PROGRAM MAIN
VAR
END_VAR

//Tc3_Motion.WareHousingExample_Tc3_DriveMotionControl();

WareHousingExample_Tc3_DriveMotionControl();

END_PROGRAM

(* stored: Version 1.1.0.1, ProductVersion 3.1.4024.12
   POU MAIN: Id {e3bb108d-9a15-4605-b94f-cc9939549109}, SpecialFunc None *)
